# EPICS autosave request: iocBoot/gmca_23b_ioc2/dbSave/XY_P1_.req
%
% BURT Request File
%
% $(P)XY:P1:  X-Y positioner #1
%

file assy.req ASSY=$(P)XY:P1
file mtr1.req MTR1=$(P)XY:mx1
file mtr1.req MTR1=$(P)XY:my1
file drv1.req DRV1=$(P)XY:X1
file drv1.req DRV1=$(P)XY:Y1
